PROGRAM MAIN
VAR
	Controller: FB_Controller;
END_VAR

Controller();

END_PROGRAM

(* stored: Version 1.1.0.1, ProductVersion 3.1.4024.6
   POU MAIN: Id {b429125e-3b4d-48ba-ac23-7b0d09072c1b}, SpecialFunc None *)
